INTERFACE I_Event

METHOD PUBLIC M_Critical : BOOL
VAR_INPUT
	nID:				UDINT;
	sMessage:			STRING(255);
END_VAR
END_METHOD

METHOD PUBLIC M_Error : BOOL
VAR_INPUT
	nID:				UDINT;
	sMessage:			STRING(255);
END_VAR
END_METHOD

METHOD PUBLIC M_Info : BOOL
VAR_INPUT
	nID:				UDINT;
	sMessage:			STRING(255);
END_VAR
END_METHOD

METHOD M_Reset : BOOL
VAR_INPUT
END_VAR
END_METHOD

METHOD PUBLIC M_Verbose : BOOL
VAR_INPUT
	sMessage:			STRING(255);
END_VAR
END_METHOD

METHOD PUBLIC M_Warning : BOOL
VAR_INPUT
	nID:				UDINT;
	sMessage:			STRING(255);
END_VAR
END_METHOD

PROPERTY PUBLIC P_Argument : I_Argument
GET
END_GET
END_PROPERTY

PROPERTY PUBLIC P_Logger : I_Logger
GET
END_GET
SET
END_SET
END_PROPERTY

END_INTERFACE

(* stored: Version 1.1.0.1
   Itf I_Event: Id {ec343ea8-6c81-46a2-a502-db967531265d}
   Method M_Critical: Id {d0c46115-ac72-4277-9bcb-ddcf7e3d7ab4}
   Method M_Error: Id {c094c3d2-f3e1-45d9-923d-9b2e1892dfd7}
   Method M_Info: Id {0cdab1e1-7612-435a-9f36-4662c49c13a4}
   Method M_Reset: Id {0b189a50-27aa-49f7-90f5-20055e5adc34}
   Method M_Verbose: Id {b412bfba-2470-494c-bd5a-84fb67b788ff}
   Method M_Warning: Id {25d7ea16-bfc2-4298-bc2f-eb93105fccab}
   Property P_Argument: Id {4316dac3-f428-4613-b61e-a2d56083c4db}
   Get Get: Id {22806bbd-7675-4908-bdec-75caf88b8e4f}
   Property P_Logger: Id {f3108a54-ddb7-4e8b-a849-4dcac1444404}
   Get Get: Id {ce49d412-fffa-4edc-87bc-4ab9c5371f4b}
   Set Set: Id {8c043879-cb58-41a7-9bfc-487118bd6496} *)
